Omron CX-Programmer project NewProject (CX-Programmer 9.75)

# PLC OMRON: CP1E N30

## Global symbols (name address type ; comment)
T000 BOOL  ; T0
T001 BOOL  ; T1
T002 BOOL  ; T2
T003 BOOL  ; T3
GREEN_A 100.01 BOOL  ; 100.01

## Program NewProgram1 (cyclic task 0)
Local symbols
GREEN_B 100.04 BOOL  ; 100.04
GreenA 100.01 BOOL  ; 100.01
MPS 100.00 BOOL  ; 100.00
RedA 100.03 BOOL  ; 100.03
RedB 100.06 BOOL  ; 100.06
Start 0.00 BOOL  ; 0.00
Stop 0.01 BOOL  ; 0.01
YellowA 100.02 BOOL  ; 100.02
YellowB 100.05 BOOL  ; 100.05

### Section Section1

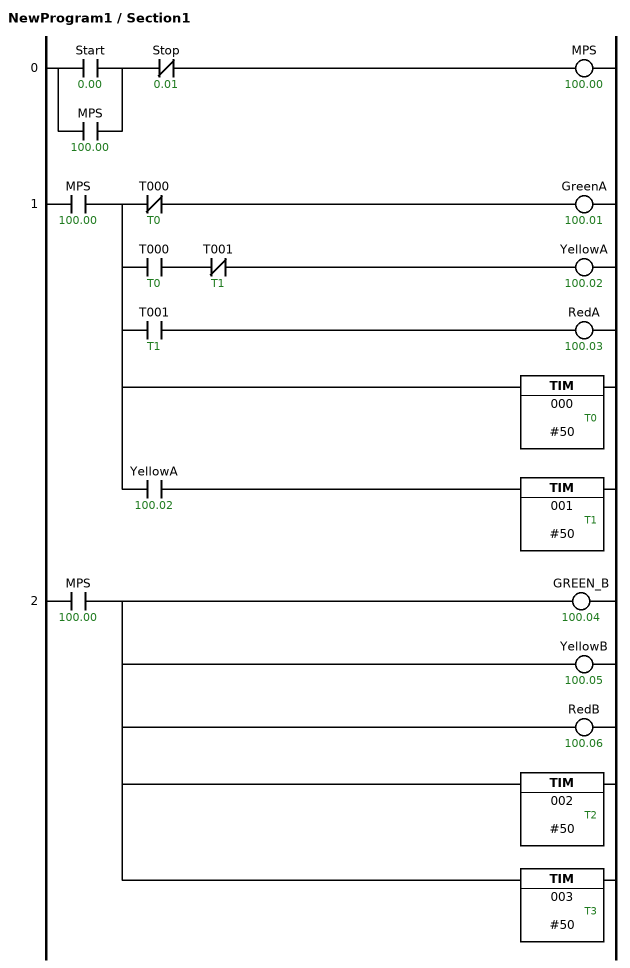
; rung 0
LD Start  ; 0.00
OR MPS  ; 100.00
ANDNOT Stop  ; 0.01
OUT MPS  ; 100.00
; rung 1
LD MPS  ; 100.00
OUT TR0
ANDNOT T000  ; T0
OUT GreenA  ; 100.01
LD TR0
AND T000  ; T0
ANDNOT T001  ; T1
OUT YellowA  ; 100.02
LD TR0
AND T001  ; T1
OUT RedA  ; 100.03
LD TR0
TIM 000 #50  ; T0
AND YellowA  ; 100.02
TIM 001 #50  ; T1
; rung 2
LD MPS  ; 100.00
OUT GREEN_B  ; 100.04
OUT YellowB  ; 100.05
OUT RedB  ; 100.06
TIM 002 #50  ; T2
TIM 003 #50  ; T3

### Section END
; rung 0
END(001)